// TIA Portal V17 export
// export: Created 2025-08-05T09:35:56.6545695Z, ExportSetting WithDefaults, DisplayName Totally Integrated Automation Portal, DisplayVersion V17, DisplayName TIA Portal Openness, DisplayVersion V17, DisplayName TIA Portal Version Control Interface, DisplayVersion V17, DisplayName SINAMICS Startdrive Advanced, DisplayVersion V17, DisplayName SINAMICS Startdrive G130, G150, S120, S150, SINAMICS MV, S210, DisplayVersion V17, DisplayName SINAMICS Startdrive G110M, G120, G120C, G120D, G120P, G115D, DisplayVersion V17, DisplayName STEP 7 Professional, DisplayVersion V17, DisplayName STEP 7 Safety, DisplayVersion V17, DisplayName WinCC Advanced, DisplayVersion V17
FUNCTION_BLOCK "Graph_Sequence"   // FB265, GRAPH
VERSION : 0.1
// stored: AcknowledgeErrorsRequired true, AutoNumber true, GraphVersion 6.0, InitialValuesAcquisition false, IsIECCheckEnabled false, LanguageInNetworks LAD, LockOperatingMode false, PermanentILProcessingInMANMode false, SetENOAutomatically false, SkipSteps true, UDAEnableTagReadback false, WithAlarmHandling true
   // inherited from GRAPH_BASE
   VAR
      OFF_SQ_BASE : Bool;
   END_VAR
   VAR_INPUT
      ACK_EF { ExternalAccessible := 'False'; ExternalVisible := 'False'; ExternalWritable := 'False'} : Bool := false;   // Acknowledge all errors and faults
      INIT_SQ { ExternalAccessible := 'False'; ExternalVisible := 'False'; ExternalWritable := 'False'} : Bool := false;   // Set sequence to initial state
      stepTimeOutTime : Time;
      iInstance_Index : DInt;
   END_VAR
   VAR_IN_OUT
      funcGrp : "typeCaCgFg";   // Funktionsgruppe / Function Group
      fgControlGeneral_1 : "typeFgControlGeneral";   // Funktionsgruppe Steuerung / Function group control system
      ioJobSelect : Int;
   END_VAR
   VAR
      instGraphEval { ExternalAccessible := 'False'; ExternalVisible := 'False'; ExternalWritable := 'False'} : "GraphEvaluation";   // FG Laser 1: S7-Graph Auswertung / FG laser 1: S7-Graph evaluation
      fgControlGeneral { ExternalAccessible := 'False'; ExternalVisible := 'False'; ExternalWritable := 'False'} : "typeFgControlGeneral";   // Funktionsgruppe Steuerung / Function group control system
      stepTimeOut : Bool;
   END_VAR
BEGIN
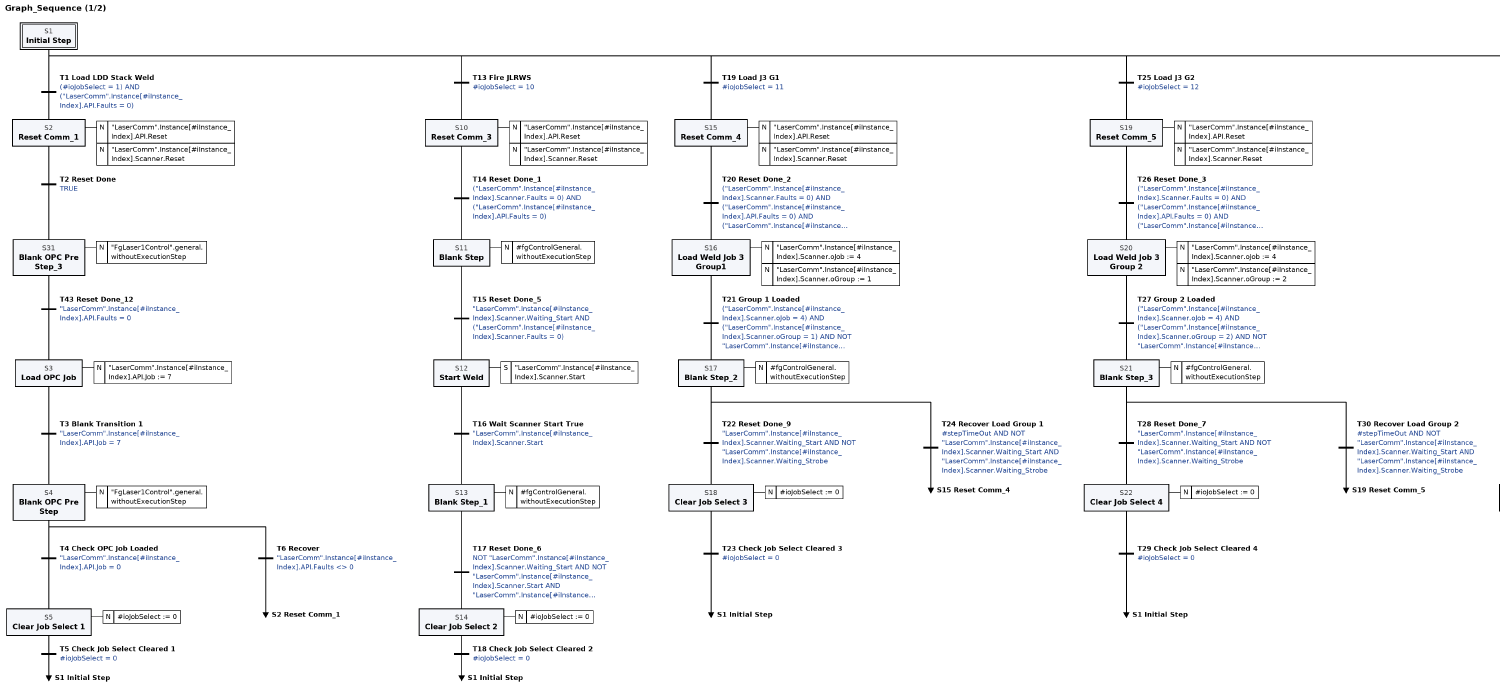
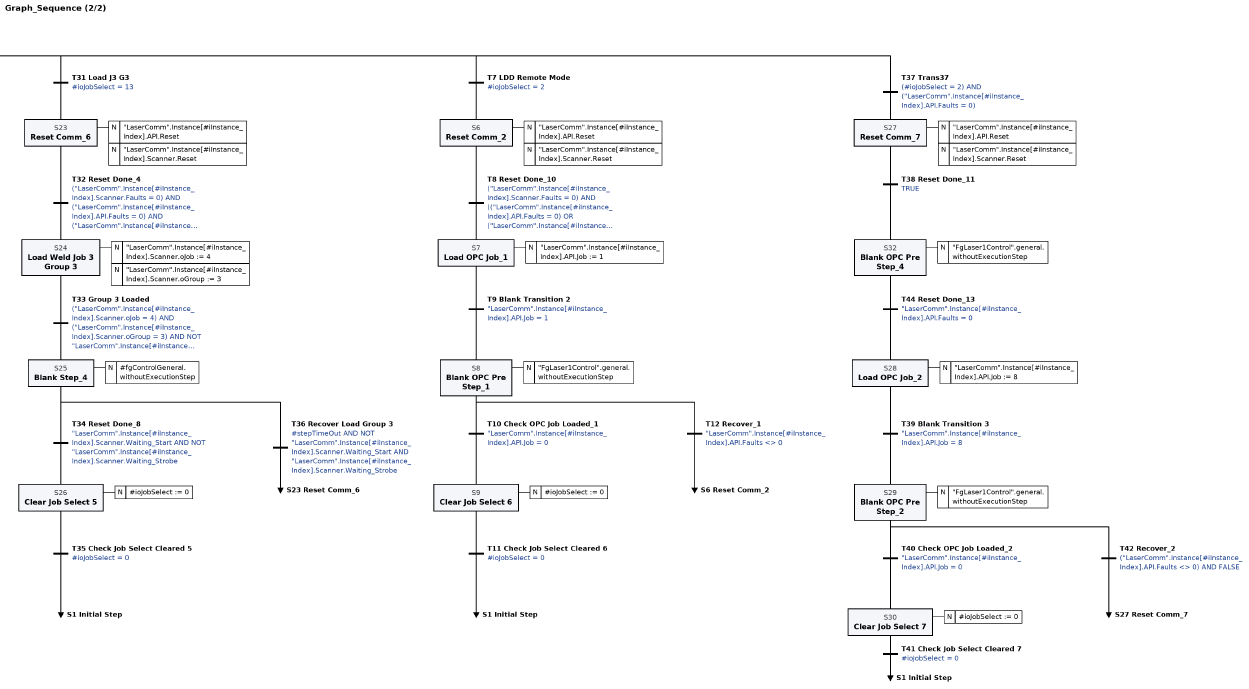
   // sequencer 1: Weld Graph Sequences
   INITIAL_STEP "Initial Step":   // S1, max time T#10S, warning time T#7S
   END_STEP
   TRANSITION "Load LDD Stack Weld" FROM "Initial Step" TO "Reset Comm_1"   // T1
      := (#ioJobSelect = 1) AND ("LaserComm".Instance[#iInstance_Index].API.Faults = 0);
   END_TRANSITION
   TRANSITION "Fire JLRWS" FROM "Initial Step" TO "Reset Comm_3"   // T13
      := #ioJobSelect = 10;
   END_TRANSITION
   TRANSITION "Load J3 G1" FROM "Initial Step" TO "Reset Comm_4"   // T19
      := #ioJobSelect = 11;
   END_TRANSITION
   TRANSITION "Load J3 G2" FROM "Initial Step" TO "Reset Comm_5"   // T25
      := #ioJobSelect = 12;
   END_TRANSITION
   TRANSITION "Load J3 G3" FROM "Initial Step" TO "Reset Comm_6"   // T31
      := #ioJobSelect = 13;
   END_TRANSITION
   TRANSITION "LDD Remote Mode" FROM "Initial Step" TO "Reset Comm_2"   // T7
      := #ioJobSelect = 2;
   END_TRANSITION
   TRANSITION Trans37 FROM "Initial Step" TO "Reset Comm_7"   // T37
      := (#ioJobSelect = 2) AND ("LaserComm".Instance[#iInstance_Index].API.Faults = 0);
   END_TRANSITION
   STEP "Reset Comm_1":   // S2, max time T#10S, warning time T#7S
      supervision V := #stepTimeOut;
              N    "LaserComm".Instance[#iInstance_Index].API.Reset
              N    "LaserComm".Instance[#iInstance_Index].Scanner.Reset
   END_STEP
   TRANSITION "Reset Done" FROM "Reset Comm_1" TO "Blank OPC Pre Step_3"   // T2
      := TRUE;
   END_TRANSITION
   STEP "Blank Step":   // S11, max time T#10S, warning time T#7S
      supervision V := #stepTimeOut;
              N    #fgControlGeneral.withoutExecutionStep
   END_STEP
   TRANSITION "Reset Done_5" FROM "Blank Step" TO "Start Weld"   // T15
      := "LaserComm".Instance[#iInstance_Index].Scanner.Waiting_Start AND ("LaserComm".Instance[#iInstance_Index].Scanner.Faults = 0);
   END_TRANSITION
   STEP "Clear Job Select 4":   // S22, max time T#10S, warning time T#7S
      supervision V := #stepTimeOut;
      // Clear Job Select
              N    #ioJobSelect := 0
   END_STEP
   TRANSITION "Check Job Select Cleared 4" FROM "Clear Job Select 4" TO "Initial Step"   // T29, jump: Check Jo Select Cleared
      := #ioJobSelect = 0;
   END_TRANSITION
   STEP "Clear Job Select 5":   // S26, max time T#10S, warning time T#7S
      supervision V := #stepTimeOut;
      // Clear Job Select
              N    #ioJobSelect := 0
   END_STEP
   TRANSITION "Check Job Select Cleared 5" FROM "Clear Job Select 5" TO "Initial Step"   // T35, jump: Check Jo Select Cleared
      := #ioJobSelect = 0;
   END_TRANSITION
   STEP "Load Weld Job 3 Group 3":   // S24, max time T#10S, warning time T#7S
      supervision V := #stepTimeOut;
              N    "LaserComm".Instance[#iInstance_Index].Scanner.oJob := 4
              N    "LaserComm".Instance[#iInstance_Index].Scanner.oGroup := 3
   END_STEP
   TRANSITION "Group 3 Loaded" FROM "Load Weld Job 3 Group 3" TO "Blank Step_4"   // T33
      := ("LaserComm".Instance[#iInstance_Index].Scanner.oJob = 4) AND ("LaserComm".Instance[#iInstance_Index].Scanner.oGroup = 3) AND NOT "LaserComm".Instance[#iInstance_Index].Scanner.Waiting_Strobe;
   END_TRANSITION
   STEP "Load OPC Job":   // S3, max time T#10S, warning time T#7S
      supervision V := #stepTimeOut;
              N    "LaserComm".Instance[#iInstance_Index].API.Job := 7
   END_STEP
   TRANSITION "Blank Transition 1" FROM "Load OPC Job" TO "Blank OPC Pre Step"   // T3
      := "LaserComm".Instance[#iInstance_Index].API.Job = 7;
   END_TRANSITION
   STEP "Blank OPC Pre Step":   // S4, max time T#10S, warning time T#7S
      supervision V := #stepTimeOut;
              N    "FgLaser1Control".general.withoutExecutionStep
   END_STEP
   TRANSITION "Check OPC Job Loaded" FROM "Blank OPC Pre Step" TO "Clear Job Select 1"   // T4
      := "LaserComm".Instance[#iInstance_Index].API.Job = 0;
   END_TRANSITION
   TRANSITION Recover FROM "Blank OPC Pre Step" TO "Reset Comm_1"   // T6, jump
      := "LaserComm".Instance[#iInstance_Index].API.Faults <> 0;
   END_TRANSITION
   STEP "Clear Job Select 1":   // S5, max time T#10S, warning time T#7S
      supervision V := #stepTimeOut;
      // Clear Job Select
              N    #ioJobSelect := 0
   END_STEP
   TRANSITION "Check Job Select Cleared 1" FROM "Clear Job Select 1" TO "Initial Step"   // T5, jump: Check Jo Select Cleared
      := #ioJobSelect = 0;
   END_TRANSITION
   STEP "Blank Step_1":   // S13, max time T#10S, warning time T#7S
      supervision V := #stepTimeOut;
              N    #fgControlGeneral.withoutExecutionStep
   END_STEP
   TRANSITION "Reset Done_6" FROM "Blank Step_1" TO "Clear Job Select 2"   // T17
      := NOT "LaserComm".Instance[#iInstance_Index].Scanner.Waiting_Start AND NOT "LaserComm".Instance[#iInstance_Index].Scanner.Start AND "LaserComm".Instance[#iInstance_Index].Scanner.Waiting_Strobe AND ("LaserComm".Instance[#iInstance_Index].Scanner.Faults = 0);
   END_TRANSITION
   STEP "Reset Comm_3":   // S10, max time T#10S, warning time T#7S
      supervision V := #stepTimeOut;
              N    "LaserComm".Instance[#iInstance_Index].API.Reset
              N    "LaserComm".Instance[#iInstance_Index].Scanner.Reset
   END_STEP
   TRANSITION "Reset Done_1" FROM "Reset Comm_3" TO "Blank Step"   // T14
      := ("LaserComm".Instance[#iInstance_Index].Scanner.Faults = 0) AND ("LaserComm".Instance[#iInstance_Index].API.Faults = 0);
   END_TRANSITION
   STEP "Load Weld Job 3 Group1":   // S16, max time T#10S, warning time T#7S
      supervision V := #stepTimeOut;
              N    "LaserComm".Instance[#iInstance_Index].Scanner.oJob := 4
              N    "LaserComm".Instance[#iInstance_Index].Scanner.oGroup := 1
   END_STEP
   TRANSITION "Group 1 Loaded" FROM "Load Weld Job 3 Group1" TO "Blank Step_2"   // T21
      := ("LaserComm".Instance[#iInstance_Index].Scanner.oJob = 4) AND ("LaserComm".Instance[#iInstance_Index].Scanner.oGroup = 1) AND NOT "LaserComm".Instance[#iInstance_Index].Scanner.Waiting_Strobe;
   END_TRANSITION
   STEP "Load Weld Job 3 Group 2":   // S20, max time T#10S, warning time T#7S
      supervision V := #stepTimeOut;
              N    "LaserComm".Instance[#iInstance_Index].Scanner.oJob := 4
              N    "LaserComm".Instance[#iInstance_Index].Scanner.oGroup := 2
   END_STEP
   TRANSITION "Group 2 Loaded" FROM "Load Weld Job 3 Group 2" TO "Blank Step_3"   // T27
      := ("LaserComm".Instance[#iInstance_Index].Scanner.oJob = 4) AND ("LaserComm".Instance[#iInstance_Index].Scanner.oGroup = 2) AND NOT "LaserComm".Instance[#iInstance_Index].Scanner.Waiting_Strobe;
   END_TRANSITION
   STEP "Reset Comm_4":   // S15, max time T#10S, warning time T#7S
      supervision V := #stepTimeOut;
              N    "LaserComm".Instance[#iInstance_Index].API.Reset
              N    "LaserComm".Instance[#iInstance_Index].Scanner.Reset
   END_STEP
   TRANSITION "Reset Done_2" FROM "Reset Comm_4" TO "Load Weld Job 3 Group1"   // T20
      := ("LaserComm".Instance[#iInstance_Index].Scanner.Faults = 0) AND ("LaserComm".Instance[#iInstance_Index].API.Faults = 0) AND ("LaserComm".Instance[#iInstance_Index].Scanner.oJob = 0) AND ("LaserComm".Instance[#iInstance_Index].Scanner.oGroup = 0) AND "LaserComm".Instance[#iInstance_Index].Scanner.Waiting_Strobe;
   END_TRANSITION
   STEP "Reset Comm_5":   // S19, max time T#10S, warning time T#7S
      supervision V := #stepTimeOut;
              N    "LaserComm".Instance[#iInstance_Index].API.Reset
              N    "LaserComm".Instance[#iInstance_Index].Scanner.Reset
   END_STEP
   TRANSITION "Reset Done_3" FROM "Reset Comm_5" TO "Load Weld Job 3 Group 2"   // T26
      := ("LaserComm".Instance[#iInstance_Index].Scanner.Faults = 0) AND ("LaserComm".Instance[#iInstance_Index].API.Faults = 0) AND ("LaserComm".Instance[#iInstance_Index].Scanner.oJob = 0) AND ("LaserComm".Instance[#iInstance_Index].Scanner.oGroup = 0);
   END_TRANSITION
   STEP "Reset Comm_6":   // S23, max time T#10S, warning time T#7S
      supervision V := #stepTimeOut;
              N    "LaserComm".Instance[#iInstance_Index].API.Reset
              N    "LaserComm".Instance[#iInstance_Index].Scanner.Reset
   END_STEP
   TRANSITION "Reset Done_4" FROM "Reset Comm_6" TO "Load Weld Job 3 Group 3"   // T32
      := ("LaserComm".Instance[#iInstance_Index].Scanner.Faults = 0) AND ("LaserComm".Instance[#iInstance_Index].API.Faults = 0) AND ("LaserComm".Instance[#iInstance_Index].Scanner.oJob = 0) AND ("LaserComm".Instance[#iInstance_Index].Scanner.oGroup = 0);
   END_TRANSITION
   STEP "Clear Job Select 3":   // S18, max time T#10S, warning time T#7S
      supervision V := #stepTimeOut;
      // Clear Job Select
              N    #ioJobSelect := 0
   END_STEP
   TRANSITION "Check Job Select Cleared 3" FROM "Clear Job Select 3" TO "Initial Step"   // T23, jump: Check Jo Select Cleared
      := #ioJobSelect = 0;
   END_TRANSITION
   STEP "Clear Job Select 2":   // S14, max time T#10S, warning time T#7S
      supervision V := #stepTimeOut;
      // Clear Job Select
              N    #ioJobSelect := 0
   END_STEP
   TRANSITION "Check Job Select Cleared 2" FROM "Clear Job Select 2" TO "Initial Step"   // T18, jump: Check Jo Select Cleared
      := #ioJobSelect = 0;
   END_TRANSITION
   STEP "Start Weld":   // S12, max time T#10S, warning time T#7S
      supervision V := #stepTimeOut;
              S    "LaserComm".Instance[#iInstance_Index].Scanner.Start
   END_STEP
   TRANSITION "Wait Scanner Start True" FROM "Start Weld" TO "Blank Step_1"   // T16
      := "LaserComm".Instance[#iInstance_Index].Scanner.Start;
   END_TRANSITION
   STEP "Blank Step_3":   // S21, max time T#10S, warning time T#7S
      supervision V := #stepTimeOut;
              N    #fgControlGeneral.withoutExecutionStep
   END_STEP
   TRANSITION "Reset Done_7" FROM "Blank Step_3" TO "Clear Job Select 4"   // T28
      := "LaserComm".Instance[#iInstance_Index].Scanner.Waiting_Start AND NOT "LaserComm".Instance[#iInstance_Index].Scanner.Waiting_Strobe;
   END_TRANSITION
   TRANSITION "Recover Load Group 2" FROM "Blank Step_3" TO "Reset Comm_5"   // T30, jump
      := #stepTimeOut AND NOT "LaserComm".Instance[#iInstance_Index].Scanner.Waiting_Start AND "LaserComm".Instance[#iInstance_Index].Scanner.Waiting_Strobe;
   END_TRANSITION
   STEP "Blank Step_4":   // S25, max time T#10S, warning time T#7S
      supervision V := #stepTimeOut;
              N    #fgControlGeneral.withoutExecutionStep
   END_STEP
   TRANSITION "Reset Done_8" FROM "Blank Step_4" TO "Clear Job Select 5"   // T34
      := "LaserComm".Instance[#iInstance_Index].Scanner.Waiting_Start AND NOT "LaserComm".Instance[#iInstance_Index].Scanner.Waiting_Strobe;
   END_TRANSITION
   TRANSITION "Recover Load Group 3" FROM "Blank Step_4" TO "Reset Comm_6"   // T36, jump
      := #stepTimeOut AND NOT "LaserComm".Instance[#iInstance_Index].Scanner.Waiting_Start AND "LaserComm".Instance[#iInstance_Index].Scanner.Waiting_Strobe;
   END_TRANSITION
   STEP "Blank Step_2":   // S17, max time T#10S, warning time T#7S
      supervision V := #stepTimeOut;
              N    #fgControlGeneral.withoutExecutionStep
   END_STEP
   TRANSITION "Reset Done_9" FROM "Blank Step_2" TO "Clear Job Select 3"   // T22
      := "LaserComm".Instance[#iInstance_Index].Scanner.Waiting_Start AND NOT "LaserComm".Instance[#iInstance_Index].Scanner.Waiting_Strobe;
   END_TRANSITION
   TRANSITION "Recover Load Group 1" FROM "Blank Step_2" TO "Reset Comm_4"   // T24, jump
      := #stepTimeOut AND NOT "LaserComm".Instance[#iInstance_Index].Scanner.Waiting_Start AND "LaserComm".Instance[#iInstance_Index].Scanner.Waiting_Strobe;
   END_TRANSITION
   STEP "Reset Comm_2":   // S6, max time T#10S, warning time T#7S
      supervision V := #stepTimeOut;
              N    "LaserComm".Instance[#iInstance_Index].API.Reset
              N    "LaserComm".Instance[#iInstance_Index].Scanner.Reset
   END_STEP
   TRANSITION "Reset Done_10" FROM "Reset Comm_2" TO "Load OPC Job_1"   // T8
      := ("LaserComm".Instance[#iInstance_Index].Scanner.Faults = 0) AND (("LaserComm".Instance[#iInstance_Index].API.Faults = 0) OR ("LaserComm".Instance[#iInstance_Index].API.Faults = 64));
   END_TRANSITION
   STEP "Load OPC Job_1":   // S7, max time T#10S, warning time T#7S
      supervision V := #stepTimeOut;
              N    "LaserComm".Instance[#iInstance_Index].API.Job := 1
   END_STEP
   TRANSITION "Blank Transition 2" FROM "Load OPC Job_1" TO "Blank OPC Pre Step_1"   // T9
      := "LaserComm".Instance[#iInstance_Index].API.Job = 1;
   END_TRANSITION
   STEP "Blank OPC Pre Step_1":   // S8, max time T#10S, warning time T#7S
      supervision V := #stepTimeOut;
              N    "FgLaser1Control".general.withoutExecutionStep
   END_STEP
   TRANSITION "Check OPC Job Loaded_1" FROM "Blank OPC Pre Step_1" TO "Clear Job Select 6"   // T10
      := "LaserComm".Instance[#iInstance_Index].API.Job = 0;
   END_TRANSITION
   TRANSITION Recover_1 FROM "Blank OPC Pre Step_1" TO "Reset Comm_2"   // T12, jump
      := "LaserComm".Instance[#iInstance_Index].API.Faults <> 0;
   END_TRANSITION
   STEP "Clear Job Select 6":   // S9, max time T#10S, warning time T#7S
      supervision V := #stepTimeOut;
      // Clear Job Select
              N    #ioJobSelect := 0
   END_STEP
   TRANSITION "Check Job Select Cleared 6" FROM "Clear Job Select 6" TO "Initial Step"   // T11, jump: Check Jo Select Cleared
      := #ioJobSelect = 0;
   END_TRANSITION
   STEP "Reset Comm_7":   // S27, max time T#10S, warning time T#7S
      supervision V := #stepTimeOut;
              N    "LaserComm".Instance[#iInstance_Index].API.Reset
              N    "LaserComm".Instance[#iInstance_Index].Scanner.Reset
   END_STEP
   TRANSITION "Reset Done_11" FROM "Reset Comm_7" TO "Blank OPC Pre Step_4"   // T38
      := TRUE;
   END_TRANSITION
   STEP "Load OPC Job_2":   // S28, max time T#10S, warning time T#7S
      supervision V := #stepTimeOut;
              N    "LaserComm".Instance[#iInstance_Index].API.Job := 8
   END_STEP
   TRANSITION "Blank Transition 3" FROM "Load OPC Job_2" TO "Blank OPC Pre Step_2"   // T39
      := "LaserComm".Instance[#iInstance_Index].API.Job = 8;
   END_TRANSITION
   STEP "Blank OPC Pre Step_2":   // S29, max time T#10S, warning time T#7S
      supervision V := #stepTimeOut;
              N    "FgLaser1Control".general.withoutExecutionStep
   END_STEP
   TRANSITION "Check OPC Job Loaded_2" FROM "Blank OPC Pre Step_2" TO "Clear Job Select 7"   // T40
      := "LaserComm".Instance[#iInstance_Index].API.Job = 0;
   END_TRANSITION
   TRANSITION Recover_2 FROM "Blank OPC Pre Step_2" TO "Reset Comm_7"   // T42, jump
      := ("LaserComm".Instance[#iInstance_Index].API.Faults <> 0) AND FALSE;
   END_TRANSITION
   STEP "Clear Job Select 7":   // S30, max time T#10S, warning time T#7S
      supervision V := #stepTimeOut;
      // Clear Job Select
              N    #ioJobSelect := 0
   END_STEP
   TRANSITION "Check Job Select Cleared 7" FROM "Clear Job Select 7" TO "Initial Step"   // T41, jump: Check Jo Select Cleared
      := #ioJobSelect = 0;
   END_TRANSITION
   STEP "Blank OPC Pre Step_3":   // S31, max time T#10S, warning time T#7S
      supervision V := #stepTimeOut;
              N    "FgLaser1Control".general.withoutExecutionStep
   END_STEP
   TRANSITION "Reset Done_12" FROM "Blank OPC Pre Step_3" TO "Load OPC Job"   // T43
      := "LaserComm".Instance[#iInstance_Index].API.Faults = 0;
   END_TRANSITION
   STEP "Blank OPC Pre Step_4":   // S32, max time T#10S, warning time T#7S
      supervision V := #stepTimeOut;
              N    "FgLaser1Control".general.withoutExecutionStep
   END_STEP
   TRANSITION "Reset Done_13" FROM "Blank OPC Pre Step_4" TO "Load OPC Job_2"   // T44
      := "LaserComm".Instance[#iInstance_Index].API.Faults = 0;
   END_TRANSITION

   // permanent post-instructions
   NETWORK 1
      #instGraphEval(rtData := #RT_DATA,   // "GraphEvaluation"
                     timeOutTime := #stepTimeOutTime,
                     funcGrp := #funcGrp,
                     fgControlGeneral := #fgControlGeneral,
                     timeOut => #stepTimeOut);
END_FUNCTION_BLOCK
